// TIA Portal V19 export
TYPE "udt_PAC3220"
// stored: Access Published
   STRUCT
      Voltage_L1 { ExternalWritable := 'False'} : Real;
      Voltage_L2 { ExternalWritable := 'False'} : Real;
      Voltage_L3 { ExternalWritable := 'False'} : Real;
      Current_L1 { ExternalWritable := 'False'} : Real;
      Current_L2 { ExternalWritable := 'False'} : Real;
      Current_L3 { ExternalWritable := 'False'} : Real;
      "AverageVoltageUL-L" { ExternalWritable := 'False'} : Real;
      AverageCurrent { ExternalWritable := 'False'} : Real;
      TotalActivePower { ExternalWritable := 'False'} : Real;
      TotalReactivePower { ExternalWritable := 'False'} : Real;
      TotalActiveEnergy { ExternalWritable := 'False'} : LReal;
      TotalApparentEnergy { ExternalWritable := 'False'} : LReal;
   END_STRUCT;
END_TYPE
